{attribute 'GeneratedUsingTerminal: EP8309-0022-0021'}
{attribute addProperty BoxType "EP8309-0022-0021"}
{attribute addProperty Id "ControlAT %Q*Control_254441A53PWM_outputAT %Q*INT2"}
{attribute addProperty CRC "1676763876"}
{attribute addProperty Size "5"}
TYPE PWM_Control_63F162E4 :
STRUCT
	{attribute addProperty Name "Control"}
	Control AT %Q* : Control_254441A5;
	{attribute addProperty Name "PWM_output"}
	PWM_output AT %Q* : INT;
END_STRUCT
END_TYPE

(* stored: Version 1.2.0.0, ProductVersion 3.1.4024.9
   DUT PWM_Control_63F162E4: Id {261d7ca5-4209-43ce-bf16-3c7f6bfb4e09} *)
